
// ===== library: MasterCopy "Copy of HMI default tag tables to HMI tags" =====

// ===== library: MasterCopy "Copy of HMI default tag tables to HMI tags_1" =====

// ===== library: MasterCopy "HMI_1" =====

(* ===== HMI "HMI_RT_1" =====
system functions are stored by id; their names below are inferred from use

graphic list "GraphList_Btn_Template_Settings": 0 'Graphic_13'; 1 'Graphic_12'

graphic list "GraphList_Proportional_Valve": 0 'Graphic_45'; 1 'Graphic_46'

graphic list "GraphList_Pump": 0 'Graphic_27'; 1 'Graphic_26'

screen "Alarm" 800x480, template "Template"
   on GenerateScreen: SetBit("_xState_Btn_Alarm")
   on ClearScreen: ResetBit("_xState_Btn_Alarm")
   AlarmView "Alarm view_1" at 5,48 size 592x422
   Button "Template_Button_4" at 600,409 size 83x58; TextOff 'Text'; PictureList "GraphList_Btn_Template_Settings"; PictureOff "Graphic_49"; PictureOn "Graphic_50"
      ProcessValue <- "_xState_Btn_Settings"
   Button "Template_Button_1" at 600,48 size 83x58; TextOff 'Text'; PictureList "GraphList_Btn_Template_Settings"; PictureOff "Graphic_54"; PictureOn "Graphic_50"
      on Release: ActivateScreen("Alarm Buffer", 0)
      ProcessValue <- "_xState_Btn_Settings"

screen "Alarm Buffer" 800x480, template "Template"
   on GenerateScreen: SetBit("_xState_Btn_Alarm_Buffer")
   on ClearScreen: ResetBit("_xState_Btn_Alarm_Buffer")
   AlarmView "Alarm view_1" at 5,48 size 592x422
   Button "Template_Button_4" at 600,49 size 83x58; TextOff 'Text'; PictureList "GraphList_Btn_Template_Settings"; PictureOff "Graphic_52"; PictureOn "Graphic_50"
      on Release: function_efd93a16()
      ProcessValue <- "_xState_Btn_Settings"

screen "Level Config" 800x480, template "Template"
   on GenerateScreen: SetBit("_xState_Btn_Level_Config")
   on ClearScreen: ResetBit("_xState_Btn_Level_Config")
   TrendView "Trend view_1" at 38,167 size 644x300
   IOField "I/O field_1" at 442,76 size 105x27; FormatPattern 999.99
   IOField "I/O field_2" at 442,105 size 105x27; FormatPattern 99.99
   IOField "I/O field_3" at 442,135 size 105x27; FormatPattern 99.99
   TextField "Text field_1" at 553,80 size 107x23; Text 'Proportional'
   TextField "Text field_2" at 552,108 size 71x23; Text 'Integral'
   TextField "Text field_3" at 552,136 size 89x23; Text 'Derivative'
   Button "Button_1" at 442,47 size 218x28; TextOff 'Save PID Parameters'
   Button "Button_2" at 299,59 size 96x45; TextOff 'Enable'
   Button "Button_5" at 299,116 size 96x41; TextOff 'Disable'
   IOField "I/O field_4" at 32,69 size 105x33; FormatPattern 999
   TextField "Text field_4" at 148,76 size 75x23; Text 'SetPoint'
   IOField "I/O field_5" at 33,112 size 105x33; FormatPattern 999
   TextField "Text field_5" at 145,118 size 118x23; Text 'Process Value'
   Button "Button_3" at 1,0 size 157x40; TextOff 'OverView'
      on Release: ActivateScreen("Level OverView", 0)
      Appearance <- "_xState_Btn_Level_Overview"
   Button "Button_4" at 162,0 size 157x40; TextOff 'Configuration'
      on Release: ActivateScreen("Level Config", 0)
      Appearance <- "_xState_Btn_Level_Config"

screen "Level OverView" 800x480, template "Template"
   on GenerateScreen: SetBit("_xState_Btn_Level_Overview")
   on ClearScreen: ResetBit("_xState_Btn_Level_Overview")
   GraphicView "Graphic view_4" at 128,89 size 150x187; Picture "Graphic_25"
   GraphicView "Graphic view_1" at 416,163 size 148x178; Picture "Graphic_25"
   GraphicView "Graphic view_21" at 319,78 size 45x23; Picture "Graphic_40"
   GraphicView "Graphic view_25" at 222,281 size 40x21; Picture "Graphic_40"
   GraphicView "Graphic view_18" at 85,270 size 31x44; Picture "Graphic_39"
   GraphicView "Graphic view_20" at 502,367 size 51x31; Picture "Graphic_40"
   Bar "Bar_1" at 140,124 size 128x115; MinimumValue 0; MaximumValue 300
      ProcessValue <- "PV"
   Button "Button_1" at 432,372 size 43x52; TextOff 'Text'; PictureList "GraphList_Pump"
   GraphicView "Graphic view_2" at 116,382 size 322x34; Picture "Graphic_28"
   GraphicView "Graphic view_7" at 81,383 size 36x32; Picture "Graphic_32"
   GraphicView "Graphic view_3" at 83,310 size 34x75; Picture "Graphic_33"
   GraphicView "Graphic view_5" at 111,211 size 30x34; Picture "Graphic_28"
   GraphicView "Graphic view_6" at 474,333 size 34x38; Picture "Graphic_33"
   GraphicView "Graphic view_8" at 474,363 size 35x41; Picture "Graphic_36"
   GraphicView "Graphic view_9" at 191,258 size 34x22; Picture "Graphic_33"
   GraphicView "Graphic view_10" at 259,275 size 173x34; Picture "Graphic_28"
   GraphicView "Graphic view_11" at 266,116 size 27x34; Picture "Graphic_28"
   GraphicView "Graphic view_12" at 357,71 size 137x34; Picture "Graphic_28"
   GraphicView "Graphic view_13" at 524,71 size 83x34; Picture "Graphic_28"
   GraphicView "Graphic view_14" at 547,187 size 59x34; Picture "Graphic_28"
   GraphicView "Graphic view_15" at 604,98 size 34x94; Picture "Graphic_33"
   GraphicView "Graphic view_16" at 194,60 size 31x41; Picture "Graphic_37"
   GraphicView "Graphic view_17" at 190,276 size 36x32; Picture "Graphic_32"
   GraphicView "Graphic view_19" at 290,114 size 37x37; Picture "Graphic_42"
   GraphicView "Graphic view_23" at 291,104 size 34x16; Picture "Graphic_33"
   GraphicView "Graphic view_24" at 292,75 size 33x31; Picture "Graphic_43"
   GraphicView "Graphic view_26" at 84,212 size 33x33; Picture "Graphic_43"
   GraphicView "Graphic view_27" at 83,241 size 34x38; Picture "Graphic_33"
   GraphicView "Graphic view_28" at 544,366 size 30x34; Picture "Graphic_28"
   GraphicView "Graphic view_29" at 603,186 size 37x37; Picture "Graphic_42"
   GraphicView "Graphic view_30" at 603,70 size 37x37; Picture "Graphic_44"
   Button "Button_2" at 491,67 size 36x41; TextOff 'Text'; PictureList "GraphList_Proportional_Valve"
   GraphicView "Graphic view_31" at 560,343 size 82x83; Picture "Graphic_48"
   Button "Button_3" at 1,0 size 157x40; TextOff 'OverView'
      Appearance <- "_xState_Btn_Level_Overview"
   Button "Button_4" at 162,0 size 157x40; TextOff 'Configuration'
      on Release: ActivateScreen("Level Config", 0)
      Appearance <- "_xState_Btn_Level_Config"
   TextField "Text field_1" at 70,162 size 45x23; Text 'S112'
   TextField "Text field_2" at 224,50 size 46x23; Text 'B102'
   TextField "Text field_3" at 340,186 size 46x23; Text 'B113'
   TextField "Text field_4" at 594,287 size 46x23; Text 'B114'
   TextField "Text field_5" at 424,140 size 45x23; Text 'S111'
   TextField "Text field_6" at 466,48 size 113x20; Text 'Proportion valve'
   TextField "Text field_7" at 115,286 size 46x23; Text 'V101'
   TextField "Text field_8" at 221,302 size 46x23; Text 'V110'
   TextField "Text field_9" at 504,396 size 46x23; Text 'V105'
   TextField "Text field_10" at 319,103 size 46x23; Text 'V112'
   TextField "Text field_11" at 508,138 size 82x20; Text 'Float switch'
   TextField "Text field_12" at 580,266 size 101x20; Text 'Low Level Cap.'
   TextField "Text field_13" at 288,165 size 103x20; Text 'High Level Cap.'
   TextField "Text field_14" at 56,141 size 82x20; Text 'Float switch'
   TextField "Text field_15" at 224,68 size 69x20; Text 'Ultrasonic'
   TextField "Text field_16" at 429,353 size 40x20; Text 'Pump'

screen "Overview" 800x480, template "Template"
   on GenerateScreen: SetBit("_xState_Btn_Overview")
   on ClearScreen: ResetBit("_xState_Btn_Overview")
   Button "Button_1" at 140,201 size 182x58; TextOff 'Level Control'; PictureOff "level_ind"
      on Release: ActivateScreen("Level OverView", 0)
   Button "Button_2" at 377,203 size 183x54; TextOff 'Flow Control'; PictureOff "level_ind"
   Button "Button_3" at 143,284 size 182x58; TextOff 'Level Control'; PictureOff "level_ind"
      on Release: ActivateScreen("Level OverView", 0)
   Button "Button_4" at 377,283 size 182x58; TextOff 'Level Control'; PictureOff "level_ind"
      on Release: ActivateScreen("Level OverView", 0)

screen "Recipe" 800x480, template "Template"
   on GenerateScreen: SetBit("_xState_Btn_Recipe")
   on ClearScreen: ResetBit("_xState_Btn_Recipe")

screen "Settings" 800x480, template "Template"
   on GenerateScreen: SetBit("_xState_Btn_Settings")
   on ClearScreen: ResetBit("_xState_Btn_Settings")
*)

(* ===== HMI "HMI_RT_1" =====
connection "HMI_Connection_1": 

HMI tags "Local Template"
   "_iScreenNumber" : Int, internal
   "_xState_Btn_Overview" : Bool, internal
   "_xState_Btn_Alarm" : Bool, internal
   "_xState_Btn_Recipe" : Bool, internal
   "_xState_Btn_Settings" : Bool, internal
   "_xState_Btn_Level_Overview" : Bool, internal
   "_xState_Btn_Level_Config" : Bool, internal
   "_xState_Btn_Alarm_Buffer" : Bool, internal

HMI tags "Default tag table"
   "Tag_ScreenNumber" : UInt, internal
   "PV" : DInt = PLC PV AT %QD42, 1 s
*)

(* ===== HMI "HMI_RT_1" =====
system functions are stored by id; their names below are inferred from use

graphic list "GraphList_Btn_Template_Recipe": 0 'Graphic_14'; 1 'Graphic_15'

graphic list "GraphList_Btn_Template_Alarm": 0 'Graphic_16'; 1 'Graphic_17'

graphic list "GraphList_Btn_Template_Settings": 0 'Graphic_13'; 1 'Graphic_12'

graphic list "GraphList_Btn_Template_Overview": 0 'Graphic_19'; 1 'Graphic_18'

Template "Template" 800x480
   Button "Template_Button_1" at 694,1 size 100x75; TextOff 'Text'; PictureList "GraphList_Btn_Template_Overview"
      on Release: ActivateScreen("Overview", 0)
      ProcessValue <- "_xState_Btn_Overview"
   Button "Template_Button_2" at 694,79 size 100x75; TextOff 'Text'; PictureList "GraphList_Btn_Template_Alarm"
      on Release: ActivateScreen("Alarm", 0)
      ProcessValue <- "_xState_Btn_Alarm"
   Button "Template_Button_3" at 694,157 size 100x75; TextOff 'Text'; PictureList "GraphList_Btn_Template_Recipe"
      on Release: ActivateScreen("Recipe", 0)
      ProcessValue <- "_xState_Btn_Recipe"
   Button "Template_Button_4" at 693,235 size 100x75; TextOff 'Text'; PictureList "GraphList_Btn_Template_Settings"
      on Release: ActivateScreen("Settings", 0)
      ProcessValue <- "_xState_Btn_Settings"
   TextField "Template_Text field_3" at 692,351 size 90x23; Text 'Start/stop'
*)

(* ===== HMI "HMI_RT_1" =====
connection "HMI_Connection_1": 

HMI tags "Local Template"
   "_iScreenNumber" : Int, internal
   "_xState_Btn_Overview" : Bool, internal
   "_xState_Btn_Alarm" : Bool, internal
   "_xState_Btn_Recipe" : Bool, internal
   "_xState_Btn_Settings" : Bool, internal
   "_xState_Btn_Level_Overview" : Bool, internal
   "_xState_Btn_Level_Config" : Bool, internal
   "_xState_Btn_Alarm_Buffer" : Bool, internal

HMI tags "Default tag table"
   "Tag_ScreenNumber" : UInt, internal
   "PV" : DInt = PLC PV AT %QD42, 1 s
*)

(* ===== HMI "HMI_RT_1" =====
system functions are stored by id; their names below are inferred from use
connection "HMI_Connection_1": ETHERNET, SMART_S7_1500_OMS

HMI tags "Local Template"
   "_iScreenNumber" : Int, internal
   "_xState_Btn_Overview" : Bool, internal
   "_xState_Btn_Alarm" : Bool, internal
   "_xState_Btn_Recipe" : Bool, internal
   "_xState_Btn_Settings" : Bool, internal
   "_xState_Btn_Level_Overview" : Bool, internal
   "_xState_Btn_Level_Config" : Bool, internal
   "_xState_Btn_Alarm_Buffer" : Bool, internal

HMI tags "Default tag table"
   "Tag_ScreenNumber" : UInt, internal
   "PV" : DInt = PLC PV AT %QD42, 1 s

graphic list "GraphList_Btn_Template_Recipe": 0 'Graphic_14'; 1 'Graphic_15'

graphic list "GraphList_Btn_Template_Overview": 0 'Graphic_19'; 1 'Graphic_18'

graphic list "GraphList_Btn_Template_Alarm": 0 'Graphic_16'; 1 'Graphic_17'

graphic list "GraphList_Pump": 0 'Graphic_27'; 1 'Graphic_26'

graphic list "GraphList_Proportional_Valve": 0 'Graphic_45'; 1 'Graphic_46'

graphic list "GraphList_Btn_Template_Settings": 0 'Graphic_13'; 1 'Graphic_12'

Template "Template" 800x480
   Button "Template_Button_1" at 694,1 size 100x75; TextOff 'Text'; PictureList "GraphList_Btn_Template_Overview"
      on Release: ActivateScreen("Overview", 0)
      ProcessValue <- "_xState_Btn_Overview"
   Button "Template_Button_2" at 694,79 size 100x75; TextOff 'Text'; PictureList "GraphList_Btn_Template_Alarm"
      on Release: ActivateScreen("Alarm", 0)
      ProcessValue <- "_xState_Btn_Alarm"
   Button "Template_Button_3" at 694,157 size 100x75; TextOff 'Text'; PictureList "GraphList_Btn_Template_Recipe"
      on Release: ActivateScreen("Recipe", 0)
      ProcessValue <- "_xState_Btn_Recipe"
   Button "Template_Button_4" at 693,235 size 100x75; TextOff 'Text'; PictureList "GraphList_Btn_Template_Settings"
      on Release: ActivateScreen("Settings", 0)
      ProcessValue <- "_xState_Btn_Settings"
   TextField "Template_Text field_3" at 692,351 size 90x23; Text 'Start/stop'

screen "Alarm" 800x480, template "Template"
   on GenerateScreen: SetBit("_xState_Btn_Alarm")
   on ClearScreen: ResetBit("_xState_Btn_Alarm")
   AlarmView "Alarm view_1" at 5,48 size 592x422
   Button "Template_Button_4" at 600,409 size 83x58; TextOff 'Text'; PictureList "GraphList_Btn_Template_Settings"; PictureOff "Graphic_49"; PictureOn "Graphic_50"
      ProcessValue <- "_xState_Btn_Settings"
   Button "Template_Button_1" at 600,48 size 83x58; TextOff 'Text'; PictureList "GraphList_Btn_Template_Settings"; PictureOff "Graphic_54"; PictureOn "Graphic_50"
      on Release: ActivateScreen("Alarm Buffer", 0)
      ProcessValue <- "_xState_Btn_Settings"

screen "Alarm Buffer" 800x480, template "Template"
   on GenerateScreen: SetBit("_xState_Btn_Alarm_Buffer")
   on ClearScreen: ResetBit("_xState_Btn_Alarm_Buffer")
   AlarmView "Alarm view_1" at 5,48 size 592x422
   Button "Template_Button_4" at 600,49 size 83x58; TextOff 'Text'; PictureList "GraphList_Btn_Template_Settings"; PictureOff "Graphic_52"; PictureOn "Graphic_50"
      on Release: function_efd93a16()
      ProcessValue <- "_xState_Btn_Settings"

screen "Level Config" 800x480, template "Template"
   on GenerateScreen: SetBit("_xState_Btn_Level_Config")
   on ClearScreen: ResetBit("_xState_Btn_Level_Config")
   TrendView "Trend view_1" at 38,167 size 644x300
   IOField "I/O field_1" at 442,76 size 105x27; FormatPattern 999.99
   IOField "I/O field_2" at 442,105 size 105x27; FormatPattern 99.99
   IOField "I/O field_3" at 442,135 size 105x27; FormatPattern 99.99
   TextField "Text field_1" at 553,80 size 107x23; Text 'Proportional'
   TextField "Text field_2" at 552,108 size 71x23; Text 'Integral'
   TextField "Text field_3" at 552,136 size 89x23; Text 'Derivative'
   Button "Button_1" at 442,47 size 218x28; TextOff 'Save PID Parameters'
   Button "Button_2" at 299,59 size 96x45; TextOff 'Enable'
   Button "Button_5" at 299,116 size 96x41; TextOff 'Disable'
   IOField "I/O field_4" at 32,69 size 105x33; FormatPattern 999
   TextField "Text field_4" at 148,76 size 75x23; Text 'SetPoint'
   IOField "I/O field_5" at 33,112 size 105x33; FormatPattern 999
   TextField "Text field_5" at 145,118 size 118x23; Text 'Process Value'
   Button "Button_3" at 1,0 size 157x40; TextOff 'OverView'
      on Release: ActivateScreen("Level OverView", 0)
      Appearance <- "_xState_Btn_Level_Overview"
   Button "Button_4" at 162,0 size 157x40; TextOff 'Configuration'
      on Release: ActivateScreen("Level Config", 0)
      Appearance <- "_xState_Btn_Level_Config"

screen "Level OverView" 800x480, template "Template"
   on GenerateScreen: SetBit("_xState_Btn_Level_Overview")
   on ClearScreen: ResetBit("_xState_Btn_Level_Overview")
   GraphicView "Graphic view_4" at 128,89 size 150x187; Picture "Graphic_25"
   GraphicView "Graphic view_1" at 416,163 size 148x178; Picture "Graphic_25"
   GraphicView "Graphic view_21" at 319,78 size 45x23; Picture "Graphic_40"
   GraphicView "Graphic view_25" at 222,281 size 40x21; Picture "Graphic_40"
   GraphicView "Graphic view_18" at 85,270 size 31x44; Picture "Graphic_39"
   GraphicView "Graphic view_20" at 502,367 size 51x31; Picture "Graphic_40"
   Bar "Bar_1" at 140,124 size 128x115; MinimumValue 0; MaximumValue 300
      ProcessValue <- "PV"
   Button "Button_1" at 432,372 size 43x52; TextOff 'Text'; PictureList "GraphList_Pump"
   GraphicView "Graphic view_2" at 116,382 size 322x34; Picture "Graphic_28"
   GraphicView "Graphic view_7" at 81,383 size 36x32; Picture "Graphic_32"
   GraphicView "Graphic view_3" at 83,310 size 34x75; Picture "Graphic_33"
   GraphicView "Graphic view_5" at 111,211 size 30x34; Picture "Graphic_28"
   GraphicView "Graphic view_6" at 474,333 size 34x38; Picture "Graphic_33"
   GraphicView "Graphic view_8" at 474,363 size 35x41; Picture "Graphic_36"
   GraphicView "Graphic view_9" at 191,258 size 34x22; Picture "Graphic_33"
   GraphicView "Graphic view_10" at 259,275 size 173x34; Picture "Graphic_28"
   GraphicView "Graphic view_11" at 266,116 size 27x34; Picture "Graphic_28"
   GraphicView "Graphic view_12" at 357,71 size 137x34; Picture "Graphic_28"
   GraphicView "Graphic view_13" at 524,71 size 83x34; Picture "Graphic_28"
   GraphicView "Graphic view_14" at 547,187 size 59x34; Picture "Graphic_28"
   GraphicView "Graphic view_15" at 604,98 size 34x94; Picture "Graphic_33"
   GraphicView "Graphic view_16" at 194,60 size 31x41; Picture "Graphic_37"
   GraphicView "Graphic view_17" at 190,276 size 36x32; Picture "Graphic_32"
   GraphicView "Graphic view_19" at 290,114 size 37x37; Picture "Graphic_42"
   GraphicView "Graphic view_23" at 291,104 size 34x16; Picture "Graphic_33"
   GraphicView "Graphic view_24" at 292,75 size 33x31; Picture "Graphic_43"
   GraphicView "Graphic view_26" at 84,212 size 33x33; Picture "Graphic_43"
   GraphicView "Graphic view_27" at 83,241 size 34x38; Picture "Graphic_33"
   GraphicView "Graphic view_28" at 544,366 size 30x34; Picture "Graphic_28"
   GraphicView "Graphic view_29" at 603,186 size 37x37; Picture "Graphic_42"
   GraphicView "Graphic view_30" at 603,70 size 37x37; Picture "Graphic_44"
   Button "Button_2" at 491,67 size 36x41; TextOff 'Text'; PictureList "GraphList_Proportional_Valve"
   GraphicView "Graphic view_31" at 560,343 size 82x83; Picture "Graphic_48"
   Button "Button_3" at 1,0 size 157x40; TextOff 'OverView'
      Appearance <- "_xState_Btn_Level_Overview"
   Button "Button_4" at 162,0 size 157x40; TextOff 'Configuration'
      on Release: ActivateScreen("Level Config", 0)
      Appearance <- "_xState_Btn_Level_Config"
   TextField "Text field_1" at 70,162 size 45x23; Text 'S112'
   TextField "Text field_2" at 224,50 size 46x23; Text 'B102'
   TextField "Text field_3" at 340,186 size 46x23; Text 'B113'
   TextField "Text field_4" at 594,287 size 46x23; Text 'B114'
   TextField "Text field_5" at 424,140 size 45x23; Text 'S111'
   TextField "Text field_6" at 466,48 size 113x20; Text 'Proportion valve'
   TextField "Text field_7" at 115,286 size 46x23; Text 'V101'
   TextField "Text field_8" at 221,302 size 46x23; Text 'V110'
   TextField "Text field_9" at 504,396 size 46x23; Text 'V105'
   TextField "Text field_10" at 319,103 size 46x23; Text 'V112'
   TextField "Text field_11" at 508,138 size 82x20; Text 'Float switch'
   TextField "Text field_12" at 580,266 size 101x20; Text 'Low Level Cap.'
   TextField "Text field_13" at 288,165 size 103x20; Text 'High Level Cap.'
   TextField "Text field_14" at 56,141 size 82x20; Text 'Float switch'
   TextField "Text field_15" at 224,68 size 69x20; Text 'Ultrasonic'
   TextField "Text field_16" at 429,353 size 40x20; Text 'Pump'

screen "Overview" 800x480, template "Template"
   on GenerateScreen: SetBit("_xState_Btn_Overview")
   on ClearScreen: ResetBit("_xState_Btn_Overview")
   Button "Button_1" at 140,201 size 182x58; TextOff 'Level Control'; PictureOff "level_ind"
      on Release: ActivateScreen("Level OverView", 0)
   Button "Button_2" at 377,203 size 183x54; TextOff 'Flow Control'; PictureOff "level_ind"
   Button "Button_3" at 143,284 size 182x58; TextOff 'Level Control'; PictureOff "level_ind"
      on Release: ActivateScreen("Level OverView", 0)
   Button "Button_4" at 377,283 size 182x58; TextOff 'Level Control'; PictureOff "level_ind"
      on Release: ActivateScreen("Level OverView", 0)

screen "Recipe" 800x480, template "Template"
   on GenerateScreen: SetBit("_xState_Btn_Recipe")
   on ClearScreen: ResetBit("_xState_Btn_Recipe")

screen "Settings" 800x480, template "Template"
   on GenerateScreen: SetBit("_xState_Btn_Settings")
   on ClearScreen: ResetBit("_xState_Btn_Settings")
*)